// TIA Portal V20 export
ORGANIZATION_BLOCK "Main"   // OB1, LAD, ProgramCycle
TITLE = "Main Program Sweep (Cycle)"
{ S7_Optimized_Access := 'TRUE' }
// stored: SetENOAutomatically false
   VAR_INPUT
      Initial_Call : Bool;   // Initial call of this OB
      Remanence : Bool;   // =True, if remanent data are available
   END_VAR
BEGIN

REGION Network 1
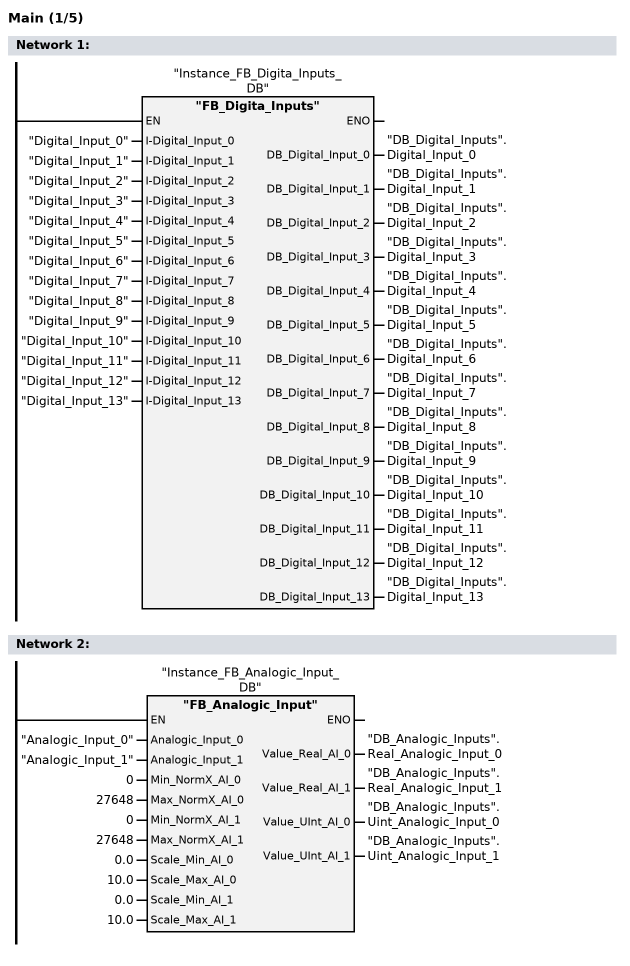
   RUNG wire#powerrail
      "Instance_FB_Digita_Inputs_DB"("I-Digital_Input_0" := "Digital_Input_0", "I-Digital_Input_1" := "Digital_Input_1", "I-Digital_Input_2" := "Digital_Input_2", "I-Digital_Input_3" := "Digital_Input_3", "I-Digital_Input_4" := "Digital_Input_4", "I-Digital_Input_5" := "Digital_Input_5", "I-Digital_Input_6" := "Digital_Input_6", "I-Digital_Input_7" := "Digital_Input_7", "I-Digital_Input_8" := "Digital_Input_8", "I-Digital_Input_9" := "Digital_Input_9", "I-Digital_Input_10" := "Digital_Input_10", "I-Digital_Input_11" := "Digital_Input_11", "I-Digital_Input_12" := "Digital_Input_12", "I-Digital_Input_13" := "Digital_Input_13", DB_Digital_Input_0 => "DB_Digital_Inputs".Digital_Input_0, DB_Digital_Input_1 => "DB_Digital_Inputs".Digital_Input_1, DB_Digital_Input_2 => "DB_Digital_Inputs".Digital_Input_2, DB_Digital_Input_3 => "DB_Digital_Inputs".Digital_Input_3, DB_Digital_Input_4 => "DB_Digital_Inputs".Digital_Input_4, DB_Digital_Input_5 => "DB_Digital_Inputs".Digital_Input_5, DB_Digital_Input_6 => "DB_Digital_Inputs".Digital_Input_6, DB_Digital_Input_7 => "DB_Digital_Inputs".Digital_Input_7, DB_Digital_Input_8 => "DB_Digital_Inputs".Digital_Input_8, DB_Digital_Input_9 => "DB_Digital_Inputs".Digital_Input_9, DB_Digital_Input_10 => "DB_Digital_Inputs".Digital_Input_10, DB_Digital_Input_11 => "DB_Digital_Inputs".Digital_Input_11, DB_Digital_Input_12 => "DB_Digital_Inputs".Digital_Input_12, DB_Digital_Input_13 => "DB_Digital_Inputs".Digital_Input_13)
   END_RUNG
   // the same network as SCL:
   "Instance_FB_Digita_Inputs_DB"("I-Digital_Input_0" := "Digital_Input_0",   // "FB_Digita_Inputs"
                           "I-Digital_Input_1" := "Digital_Input_1",
                           "I-Digital_Input_2" := "Digital_Input_2",
                           "I-Digital_Input_3" := "Digital_Input_3",
                           "I-Digital_Input_4" := "Digital_Input_4",
                           "I-Digital_Input_5" := "Digital_Input_5",
                           "I-Digital_Input_6" := "Digital_Input_6",
                           "I-Digital_Input_7" := "Digital_Input_7",
                           "I-Digital_Input_8" := "Digital_Input_8",
                           "I-Digital_Input_9" := "Digital_Input_9",
                           "I-Digital_Input_10" := "Digital_Input_10",
                           "I-Digital_Input_11" := "Digital_Input_11",
                           "I-Digital_Input_12" := "Digital_Input_12",
                           "I-Digital_Input_13" := "Digital_Input_13",
                           DB_Digital_Input_0 => "DB_Digital_Inputs".Digital_Input_0,
                           DB_Digital_Input_1 => "DB_Digital_Inputs".Digital_Input_1,
                           DB_Digital_Input_2 => "DB_Digital_Inputs".Digital_Input_2,
                           DB_Digital_Input_3 => "DB_Digital_Inputs".Digital_Input_3,
                           DB_Digital_Input_4 => "DB_Digital_Inputs".Digital_Input_4,
                           DB_Digital_Input_5 => "DB_Digital_Inputs".Digital_Input_5,
                           DB_Digital_Input_6 => "DB_Digital_Inputs".Digital_Input_6,
                           DB_Digital_Input_7 => "DB_Digital_Inputs".Digital_Input_7,
                           DB_Digital_Input_8 => "DB_Digital_Inputs".Digital_Input_8,
                           DB_Digital_Input_9 => "DB_Digital_Inputs".Digital_Input_9,
                           DB_Digital_Input_10 => "DB_Digital_Inputs".Digital_Input_10,
                           DB_Digital_Input_11 => "DB_Digital_Inputs".Digital_Input_11,
                           DB_Digital_Input_12 => "DB_Digital_Inputs".Digital_Input_12,
                           DB_Digital_Input_13 => "DB_Digital_Inputs".Digital_Input_13);
END_REGION

REGION Network 2
   RUNG wire#powerrail
      "Instance_FB_Analogic_Input_DB"(Analogic_Input_0 := "Analogic_Input_0", Analogic_Input_1 := "Analogic_Input_1", Min_NormX_AI_0 := 0, Max_NormX_AI_0 := 27648, Min_NormX_AI_1 := 0, Max_NormX_AI_1 := 27648, Scale_Min_AI_0 := 0.0, Scale_Max_AI_0 := 10.0, Scale_Min_AI_1 := 0.0, Scale_Max_AI_1 := 10.0, Value_Real_AI_0 => "DB_Analogic_Inputs".Real_Analogic_Input_0, Value_Real_AI_1 => "DB_Analogic_Inputs".Real_Analogic_Input_1, Value_UInt_AI_0 => "DB_Analogic_Inputs".Uint_Analogic_Input_0, Value_UInt_AI_1 => "DB_Analogic_Inputs".Uint_Analogic_Input_1)
   END_RUNG
   // the same network as SCL:
   "Instance_FB_Analogic_Input_DB"(Analogic_Input_0 := "Analogic_Input_0",   // "FB_Analogic_Input"
                           Analogic_Input_1 := "Analogic_Input_1",
                           Min_NormX_AI_0 := 0,
                           Max_NormX_AI_0 := 27648,
                           Min_NormX_AI_1 := 0,
                           Max_NormX_AI_1 := 27648,
                           Scale_Min_AI_0 := 0.0,
                           Scale_Max_AI_0 := 10.0,
                           Scale_Min_AI_1 := 0.0,
                           Scale_Max_AI_1 := 10.0,
                           Value_Real_AI_0 => "DB_Analogic_Inputs".Real_Analogic_Input_0,
                           Value_Real_AI_1 => "DB_Analogic_Inputs".Real_Analogic_Input_1,
                           Value_UInt_AI_0 => "DB_Analogic_Inputs".Uint_Analogic_Input_0,
                           Value_UInt_AI_1 => "DB_Analogic_Inputs".Uint_Analogic_Input_1);
END_REGION

REGION Network 3
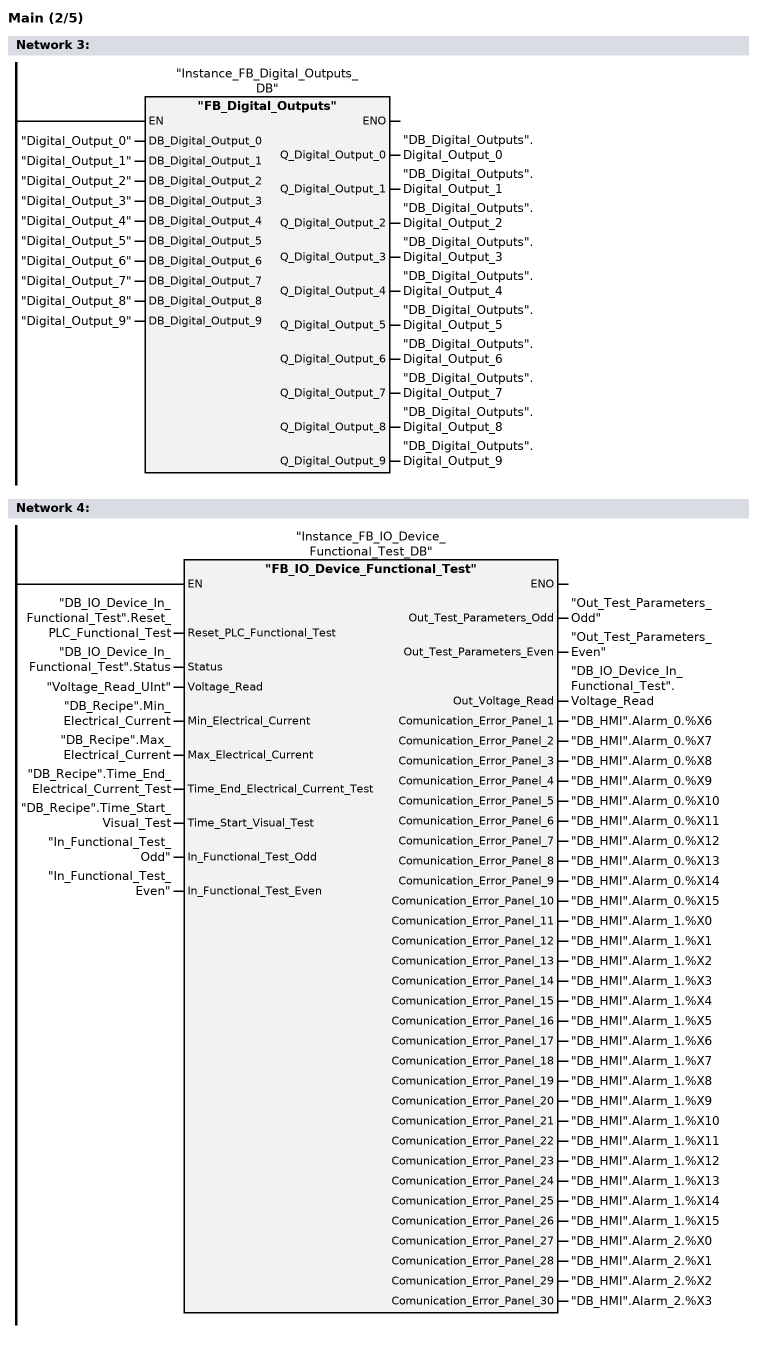
   RUNG wire#powerrail
      "Instance_FB_Digital_Outputs_DB"(DB_Digital_Output_0 := "Digital_Output_0", DB_Digital_Output_1 := "Digital_Output_1", DB_Digital_Output_2 := "Digital_Output_2", DB_Digital_Output_3 := "Digital_Output_3", DB_Digital_Output_4 := "Digital_Output_4", DB_Digital_Output_5 := "Digital_Output_5", DB_Digital_Output_6 := "Digital_Output_6", DB_Digital_Output_7 := "Digital_Output_7", DB_Digital_Output_8 := "Digital_Output_8", DB_Digital_Output_9 := "Digital_Output_9", Q_Digital_Output_0 => "DB_Digital_Outputs".Digital_Output_0, Q_Digital_Output_1 => "DB_Digital_Outputs".Digital_Output_1, Q_Digital_Output_2 => "DB_Digital_Outputs".Digital_Output_2, Q_Digital_Output_3 => "DB_Digital_Outputs".Digital_Output_3, Q_Digital_Output_4 => "DB_Digital_Outputs".Digital_Output_4, Q_Digital_Output_5 => "DB_Digital_Outputs".Digital_Output_5, Q_Digital_Output_6 => "DB_Digital_Outputs".Digital_Output_6, Q_Digital_Output_7 => "DB_Digital_Outputs".Digital_Output_7, Q_Digital_Output_8 => "DB_Digital_Outputs".Digital_Output_8, Q_Digital_Output_9 => "DB_Digital_Outputs".Digital_Output_9)
   END_RUNG
   // the same network as SCL:
   "Instance_FB_Digital_Outputs_DB"(DB_Digital_Output_0 := "Digital_Output_0",   // "FB_Digital_Outputs"
                           DB_Digital_Output_1 := "Digital_Output_1",
                           DB_Digital_Output_2 := "Digital_Output_2",
                           DB_Digital_Output_3 := "Digital_Output_3",
                           DB_Digital_Output_4 := "Digital_Output_4",
                           DB_Digital_Output_5 := "Digital_Output_5",
                           DB_Digital_Output_6 := "Digital_Output_6",
                           DB_Digital_Output_7 := "Digital_Output_7",
                           DB_Digital_Output_8 := "Digital_Output_8",
                           DB_Digital_Output_9 := "Digital_Output_9",
                           Q_Digital_Output_0 => "DB_Digital_Outputs".Digital_Output_0,
                           Q_Digital_Output_1 => "DB_Digital_Outputs".Digital_Output_1,
                           Q_Digital_Output_2 => "DB_Digital_Outputs".Digital_Output_2,
                           Q_Digital_Output_3 => "DB_Digital_Outputs".Digital_Output_3,
                           Q_Digital_Output_4 => "DB_Digital_Outputs".Digital_Output_4,
                           Q_Digital_Output_5 => "DB_Digital_Outputs".Digital_Output_5,
                           Q_Digital_Output_6 => "DB_Digital_Outputs".Digital_Output_6,
                           Q_Digital_Output_7 => "DB_Digital_Outputs".Digital_Output_7,
                           Q_Digital_Output_8 => "DB_Digital_Outputs".Digital_Output_8,
                           Q_Digital_Output_9 => "DB_Digital_Outputs".Digital_Output_9);
END_REGION

REGION Network 4
   RUNG wire#powerrail
      "Instance_FB_IO_Device_Functional_Test_DB"(Reset_PLC_Functional_Test := "DB_IO_Device_In_Functional_Test".Reset_PLC_Functional_Test, Status := "DB_IO_Device_In_Functional_Test".Status, Voltage_Read := "Voltage_Read_UInt", Min_Electrical_Current := "DB_Recipe".Min_Electrical_Current, Max_Electrical_Current := "DB_Recipe".Max_Electrical_Current, Time_End_Electrical_Current_Test := "DB_Recipe".Time_End_Electrical_Current_Test, Time_Start_Visual_Test := "DB_Recipe".Time_Start_Visual_Test, In_Functional_Test_Odd := "In_Functional_Test_Odd", In_Functional_Test_Even := "In_Functional_Test_Even", Out_Test_Parameters_Odd => "Out_Test_Parameters_Odd", Out_Test_Parameters_Even => "Out_Test_Parameters_Even", Out_Voltage_Read => "DB_IO_Device_In_Functional_Test".Voltage_Read, Comunication_Error_Panel_1 => "DB_HMI".Alarm_0.%X6, Comunication_Error_Panel_2 => "DB_HMI".Alarm_0.%X7, Comunication_Error_Panel_3 => "DB_HMI".Alarm_0.%X8, Comunication_Error_Panel_4 => "DB_HMI".Alarm_0.%X9, Comunication_Error_Panel_5 => "DB_HMI".Alarm_0.%X10, Comunication_Error_Panel_6 => "DB_HMI".Alarm_0.%X11, Comunication_Error_Panel_7 => "DB_HMI".Alarm_0.%X12, Comunication_Error_Panel_8 => "DB_HMI".Alarm_0.%X13, Comunication_Error_Panel_9 => "DB_HMI".Alarm_0.%X14, Comunication_Error_Panel_10 => "DB_HMI".Alarm_0.%X15, Comunication_Error_Panel_11 => "DB_HMI".Alarm_1.%X0, Comunication_Error_Panel_12 => "DB_HMI".Alarm_1.%X1, Comunication_Error_Panel_13 => "DB_HMI".Alarm_1.%X2, Comunication_Error_Panel_14 => "DB_HMI".Alarm_1.%X3, Comunication_Error_Panel_15 => "DB_HMI".Alarm_1.%X4, Comunication_Error_Panel_16 => "DB_HMI".Alarm_1.%X5, Comunication_Error_Panel_17 => "DB_HMI".Alarm_1.%X6, Comunication_Error_Panel_18 => "DB_HMI".Alarm_1.%X7, Comunication_Error_Panel_19 => "DB_HMI".Alarm_1.%X8, Comunication_Error_Panel_20 => "DB_HMI".Alarm_1.%X9, Comunication_Error_Panel_21 => "DB_HMI".Alarm_1.%X10, Comunication_Error_Panel_22 => "DB_HMI".Alarm_1.%X11, Comunication_Error_Panel_23 => "DB_HMI".Alarm_1.%X12, Comunication_Error_Panel_24 => "DB_HMI".Alarm_1.%X13, Comunication_Error_Panel_25 => "DB_HMI".Alarm_1.%X14, Comunication_Error_Panel_26 => "DB_HMI".Alarm_1.%X15, Comunication_Error_Panel_27 => "DB_HMI".Alarm_2.%X0, Comunication_Error_Panel_28 => "DB_HMI".Alarm_2.%X1, Comunication_Error_Panel_29 => "DB_HMI".Alarm_2.%X2, Comunication_Error_Panel_30 => "DB_HMI".Alarm_2.%X3)
   END_RUNG
   // the same network as SCL:
   "Instance_FB_IO_Device_Functional_Test_DB"(Reset_PLC_Functional_Test := "DB_IO_Device_In_Functional_Test".Reset_PLC_Functional_Test,   // "FB_IO_Device_Functional_Test"
                           Status := "DB_IO_Device_In_Functional_Test".Status,
                           Voltage_Read := "Voltage_Read_UInt",
                           Min_Electrical_Current := "DB_Recipe".Min_Electrical_Current,
                           Max_Electrical_Current := "DB_Recipe".Max_Electrical_Current,
                           Time_End_Electrical_Current_Test := "DB_Recipe".Time_End_Electrical_Current_Test,
                           Time_Start_Visual_Test := "DB_Recipe".Time_Start_Visual_Test,
                           In_Functional_Test_Odd := "In_Functional_Test_Odd",
                           In_Functional_Test_Even := "In_Functional_Test_Even",
                           Out_Test_Parameters_Odd => "Out_Test_Parameters_Odd",
                           Out_Test_Parameters_Even => "Out_Test_Parameters_Even",
                           Out_Voltage_Read => "DB_IO_Device_In_Functional_Test".Voltage_Read,
                           Comunication_Error_Panel_1 => "DB_HMI".Alarm_0.%X6,
                           Comunication_Error_Panel_2 => "DB_HMI".Alarm_0.%X7,
                           Comunication_Error_Panel_3 => "DB_HMI".Alarm_0.%X8,
                           Comunication_Error_Panel_4 => "DB_HMI".Alarm_0.%X9,
                           Comunication_Error_Panel_5 => "DB_HMI".Alarm_0.%X10,
                           Comunication_Error_Panel_6 => "DB_HMI".Alarm_0.%X11,
                           Comunication_Error_Panel_7 => "DB_HMI".Alarm_0.%X12,
                           Comunication_Error_Panel_8 => "DB_HMI".Alarm_0.%X13,
                           Comunication_Error_Panel_9 => "DB_HMI".Alarm_0.%X14,
                           Comunication_Error_Panel_10 => "DB_HMI".Alarm_0.%X15,
                           Comunication_Error_Panel_11 => "DB_HMI".Alarm_1.%X0,
                           Comunication_Error_Panel_12 => "DB_HMI".Alarm_1.%X1,
                           Comunication_Error_Panel_13 => "DB_HMI".Alarm_1.%X2,
                           Comunication_Error_Panel_14 => "DB_HMI".Alarm_1.%X3,
                           Comunication_Error_Panel_15 => "DB_HMI".Alarm_1.%X4,
                           Comunication_Error_Panel_16 => "DB_HMI".Alarm_1.%X5,
                           Comunication_Error_Panel_17 => "DB_HMI".Alarm_1.%X6,
                           Comunication_Error_Panel_18 => "DB_HMI".Alarm_1.%X7,
                           Comunication_Error_Panel_19 => "DB_HMI".Alarm_1.%X8,
                           Comunication_Error_Panel_20 => "DB_HMI".Alarm_1.%X9,
                           Comunication_Error_Panel_21 => "DB_HMI".Alarm_1.%X10,
                           Comunication_Error_Panel_22 => "DB_HMI".Alarm_1.%X11,
                           Comunication_Error_Panel_23 => "DB_HMI".Alarm_1.%X12,
                           Comunication_Error_Panel_24 => "DB_HMI".Alarm_1.%X13,
                           Comunication_Error_Panel_25 => "DB_HMI".Alarm_1.%X14,
                           Comunication_Error_Panel_26 => "DB_HMI".Alarm_1.%X15,
                           Comunication_Error_Panel_27 => "DB_HMI".Alarm_2.%X0,
                           Comunication_Error_Panel_28 => "DB_HMI".Alarm_2.%X1,
                           Comunication_Error_Panel_29 => "DB_HMI".Alarm_2.%X2,
                           Comunication_Error_Panel_30 => "DB_HMI".Alarm_2.%X3);
END_REGION

REGION Network 5
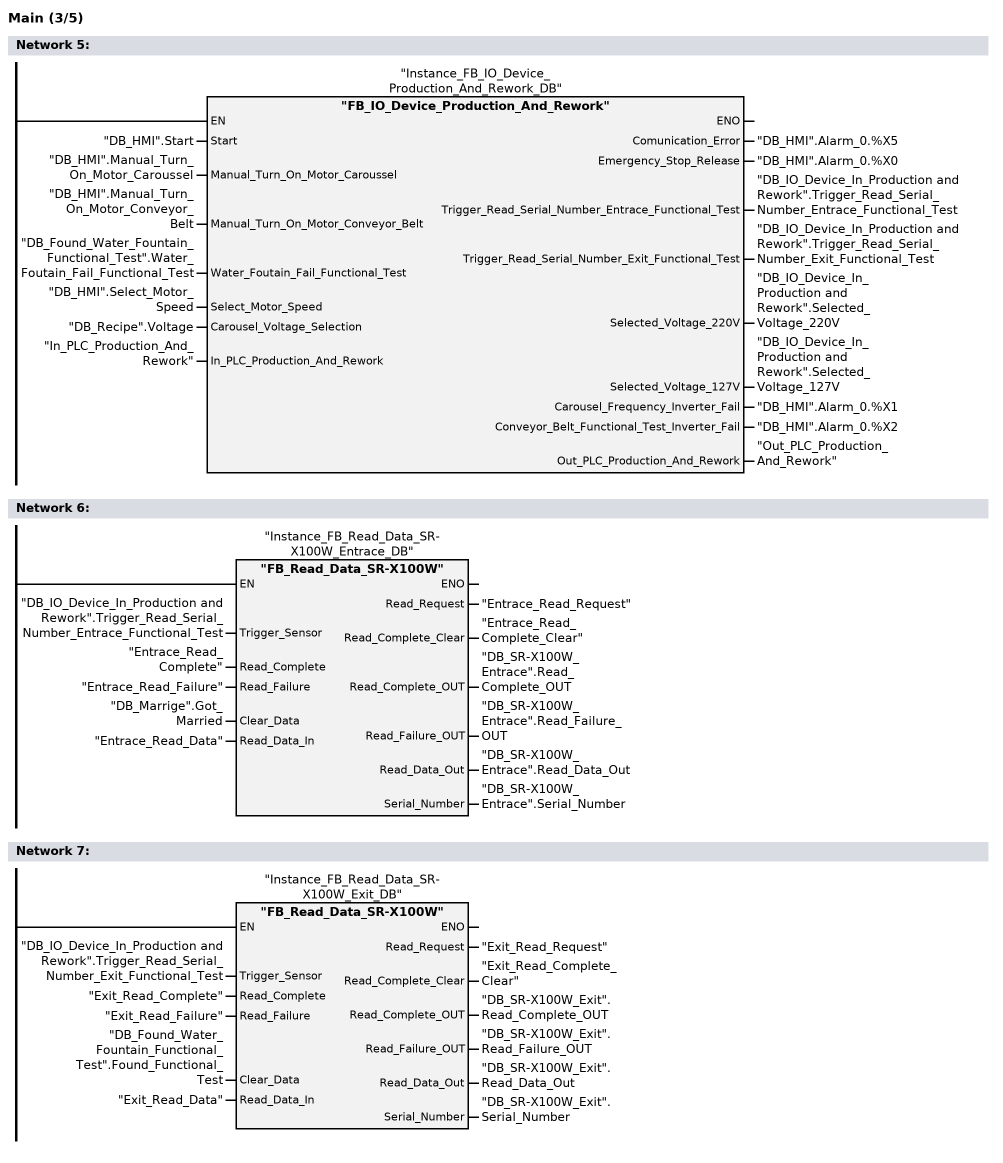
   RUNG wire#powerrail
      "Instance_FB_IO_Device_Production_And_Rework_DB"(Start := "DB_HMI".Start, Manual_Turn_On_Motor_Caroussel := "DB_HMI".Manual_Turn_On_Motor_Caroussel, Manual_Turn_On_Motor_Conveyor_Belt := "DB_HMI".Manual_Turn_On_Motor_Conveyor_Belt, Water_Foutain_Fail_Functional_Test := "DB_Found_Water_Fountain_Functional_Test".Water_Foutain_Fail_Functional_Test, Select_Motor_Speed := "DB_HMI".Select_Motor_Speed, Carousel_Voltage_Selection := "DB_Recipe".Voltage, In_PLC_Production_And_Rework := "In_PLC_Production_And_Rework", Comunication_Error => "DB_HMI".Alarm_0.%X5, Emergency_Stop_Release => "DB_HMI".Alarm_0.%X0, Trigger_Read_Serial_Number_Entrace_Functional_Test => "DB_IO_Device_In_Production and Rework".Trigger_Read_Serial_Number_Entrace_Functional_Test, Trigger_Read_Serial_Number_Exit_Functional_Test => "DB_IO_Device_In_Production and Rework".Trigger_Read_Serial_Number_Exit_Functional_Test, Selected_Voltage_220V => "DB_IO_Device_In_Production and Rework".Selected_Voltage_220V, Selected_Voltage_127V => "DB_IO_Device_In_Production and Rework".Selected_Voltage_127V, Carousel_Frequency_Inverter_Fail => "DB_HMI".Alarm_0.%X1, Conveyor_Belt_Functional_Test_Inverter_Fail => "DB_HMI".Alarm_0.%X2, Out_PLC_Production_And_Rework => "Out_PLC_Production_And_Rework")
   END_RUNG
   // the same network as SCL:
   "Instance_FB_IO_Device_Production_And_Rework_DB"(Start := "DB_HMI".Start,   // "FB_IO_Device_Production_And_Rework"
                           Manual_Turn_On_Motor_Caroussel := "DB_HMI".Manual_Turn_On_Motor_Caroussel,
                           Manual_Turn_On_Motor_Conveyor_Belt := "DB_HMI".Manual_Turn_On_Motor_Conveyor_Belt,
                           Water_Foutain_Fail_Functional_Test := "DB_Found_Water_Fountain_Functional_Test".Water_Foutain_Fail_Functional_Test,
                           Select_Motor_Speed := "DB_HMI".Select_Motor_Speed,
                           Carousel_Voltage_Selection := "DB_Recipe".Voltage,
                           In_PLC_Production_And_Rework := "In_PLC_Production_And_Rework",
                           Comunication_Error => "DB_HMI".Alarm_0.%X5,
                           Emergency_Stop_Release => "DB_HMI".Alarm_0.%X0,
                           Trigger_Read_Serial_Number_Entrace_Functional_Test => "DB_IO_Device_In_Production and Rework".Trigger_Read_Serial_Number_Entrace_Functional_Test,
                           Trigger_Read_Serial_Number_Exit_Functional_Test => "DB_IO_Device_In_Production and Rework".Trigger_Read_Serial_Number_Exit_Functional_Test,
                           Selected_Voltage_220V => "DB_IO_Device_In_Production and Rework".Selected_Voltage_220V,
                           Selected_Voltage_127V => "DB_IO_Device_In_Production and Rework".Selected_Voltage_127V,
                           Carousel_Frequency_Inverter_Fail => "DB_HMI".Alarm_0.%X1,
                           Conveyor_Belt_Functional_Test_Inverter_Fail => "DB_HMI".Alarm_0.%X2,
                           Out_PLC_Production_And_Rework => "Out_PLC_Production_And_Rework");
END_REGION

REGION Network 6
   RUNG wire#powerrail
      "Instance_FB_Read_Data_SR-X100W_Entrace_DB"(Trigger_Sensor := "DB_IO_Device_In_Production and Rework".Trigger_Read_Serial_Number_Entrace_Functional_Test, Read_Complete := "Entrace_Read_Complete", Read_Failure := "Entrace_Read_Failure", Clear_Data := "DB_Marrige".Got_Married, Read_Data_In := "Entrace_Read_Data", Read_Request => "Entrace_Read_Request", Read_Complete_Clear => "Entrace_Read_Complete_Clear", Read_Complete_OUT => "DB_SR-X100W_Entrace".Read_Complete_OUT, Read_Failure_OUT => "DB_SR-X100W_Entrace".Read_Failure_OUT, Read_Data_Out => "DB_SR-X100W_Entrace".Read_Data_Out, Serial_Number => "DB_SR-X100W_Entrace".Serial_Number)
   END_RUNG
   // the same network as SCL:
   "Instance_FB_Read_Data_SR-X100W_Entrace_DB"(Trigger_Sensor := "DB_IO_Device_In_Production and Rework".Trigger_Read_Serial_Number_Entrace_Functional_Test,   // "FB_Read_Data_SR-X100W"
                           Read_Complete := "Entrace_Read_Complete",
                           Read_Failure := "Entrace_Read_Failure",
                           Clear_Data := "DB_Marrige".Got_Married,
                           Read_Data_In := "Entrace_Read_Data",
                           Read_Request => "Entrace_Read_Request",
                           Read_Complete_Clear => "Entrace_Read_Complete_Clear",
                           Read_Complete_OUT => "DB_SR-X100W_Entrace".Read_Complete_OUT,
                           Read_Failure_OUT => "DB_SR-X100W_Entrace".Read_Failure_OUT,
                           Read_Data_Out => "DB_SR-X100W_Entrace".Read_Data_Out,
                           Serial_Number => "DB_SR-X100W_Entrace".Serial_Number);
END_REGION

REGION Network 7
   RUNG wire#powerrail
      "Instance_FB_Read_Data_SR-X100W_Exit_DB"(Trigger_Sensor := "DB_IO_Device_In_Production and Rework".Trigger_Read_Serial_Number_Exit_Functional_Test, Read_Complete := "Exit_Read_Complete", Read_Failure := "Exit_Read_Failure", Clear_Data := "DB_Found_Water_Fountain_Functional_Test".Found_Functional_Test, Read_Data_In := "Exit_Read_Data", Read_Request => "Exit_Read_Request", Read_Complete_Clear => "Exit_Read_Complete_Clear", Read_Complete_OUT => "DB_SR-X100W_Exit".Read_Complete_OUT, Read_Failure_OUT => "DB_SR-X100W_Exit".Read_Failure_OUT, Read_Data_Out => "DB_SR-X100W_Exit".Read_Data_Out, Serial_Number => "DB_SR-X100W_Exit".Serial_Number)
   END_RUNG
   // the same network as SCL:
   "Instance_FB_Read_Data_SR-X100W_Exit_DB"(Trigger_Sensor := "DB_IO_Device_In_Production and Rework".Trigger_Read_Serial_Number_Exit_Functional_Test,   // "FB_Read_Data_SR-X100W"
                           Read_Complete := "Exit_Read_Complete",
                           Read_Failure := "Exit_Read_Failure",
                           Clear_Data := "DB_Found_Water_Fountain_Functional_Test".Found_Functional_Test,
                           Read_Data_In := "Exit_Read_Data",
                           Read_Request => "Exit_Read_Request",
                           Read_Complete_Clear => "Exit_Read_Complete_Clear",
                           Read_Complete_OUT => "DB_SR-X100W_Exit".Read_Complete_OUT,
                           Read_Failure_OUT => "DB_SR-X100W_Exit".Read_Failure_OUT,
                           Read_Data_Out => "DB_SR-X100W_Exit".Read_Data_Out,
                           Serial_Number => "DB_SR-X100W_Exit".Serial_Number);
END_REGION

REGION Network 8
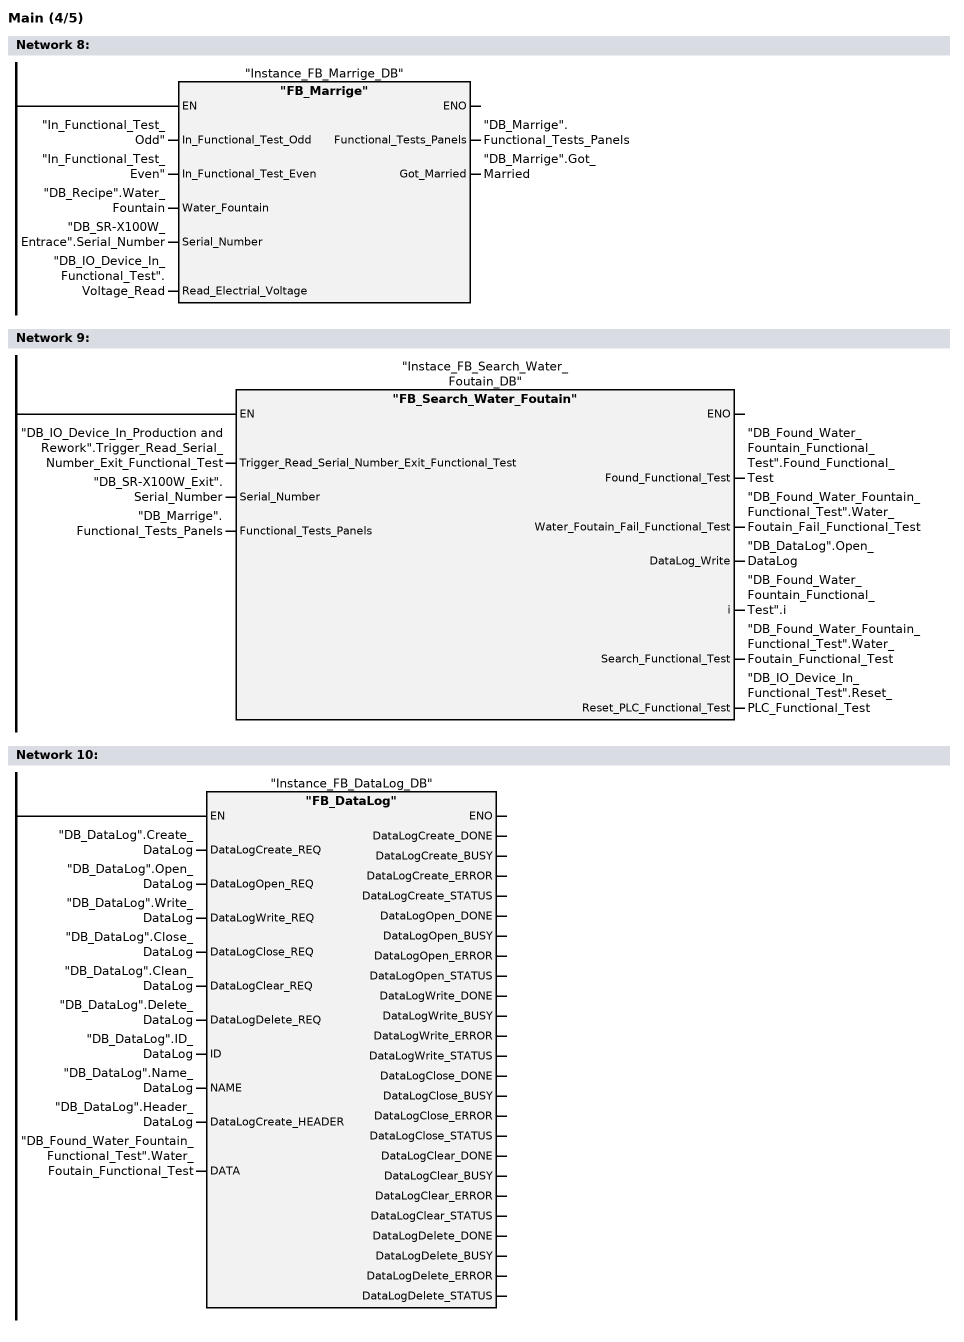
   RUNG wire#powerrail
      "Instance_FB_Marrige_DB"(In_Functional_Test_Odd := "In_Functional_Test_Odd", In_Functional_Test_Even := "In_Functional_Test_Even", Water_Fountain := "DB_Recipe".Water_Fountain, Serial_Number := "DB_SR-X100W_Entrace".Serial_Number, Read_Electrial_Voltage := "DB_IO_Device_In_Functional_Test".Voltage_Read, Functional_Tests_Panels => "DB_Marrige".Functional_Tests_Panels, Got_Married => "DB_Marrige".Got_Married)
   END_RUNG
   // the same network as SCL:
   "Instance_FB_Marrige_DB"(In_Functional_Test_Odd := "In_Functional_Test_Odd",   // "FB_Marrige"
                           In_Functional_Test_Even := "In_Functional_Test_Even",
                           Water_Fountain := "DB_Recipe".Water_Fountain,
                           Serial_Number := "DB_SR-X100W_Entrace".Serial_Number,
                           Read_Electrial_Voltage := "DB_IO_Device_In_Functional_Test".Voltage_Read,
                           Functional_Tests_Panels => "DB_Marrige".Functional_Tests_Panels,
                           Got_Married => "DB_Marrige".Got_Married);
END_REGION

REGION Network 9
   RUNG wire#powerrail
      "Instace_FB_Search_Water_Foutain_DB"(Trigger_Read_Serial_Number_Exit_Functional_Test := "DB_IO_Device_In_Production and Rework".Trigger_Read_Serial_Number_Exit_Functional_Test, Serial_Number := "DB_SR-X100W_Exit".Serial_Number, Functional_Tests_Panels := "DB_Marrige".Functional_Tests_Panels, Found_Functional_Test => "DB_Found_Water_Fountain_Functional_Test".Found_Functional_Test, Water_Foutain_Fail_Functional_Test => "DB_Found_Water_Fountain_Functional_Test".Water_Foutain_Fail_Functional_Test, DataLog_Write => "DB_DataLog".Open_DataLog, i => "DB_Found_Water_Fountain_Functional_Test".i, Search_Functional_Test => "DB_Found_Water_Fountain_Functional_Test".Water_Foutain_Functional_Test, Reset_PLC_Functional_Test => "DB_IO_Device_In_Functional_Test".Reset_PLC_Functional_Test)
   END_RUNG
   // the same network as SCL:
   "Instace_FB_Search_Water_Foutain_DB"(Trigger_Read_Serial_Number_Exit_Functional_Test := "DB_IO_Device_In_Production and Rework".Trigger_Read_Serial_Number_Exit_Functional_Test,   // "FB_Search_Water_Foutain"
                           Serial_Number := "DB_SR-X100W_Exit".Serial_Number,
                           Functional_Tests_Panels := "DB_Marrige".Functional_Tests_Panels,
                           Found_Functional_Test => "DB_Found_Water_Fountain_Functional_Test".Found_Functional_Test,
                           Water_Foutain_Fail_Functional_Test => "DB_Found_Water_Fountain_Functional_Test".Water_Foutain_Fail_Functional_Test,
                           DataLog_Write => "DB_DataLog".Open_DataLog,
                           i => "DB_Found_Water_Fountain_Functional_Test".i,
                           Search_Functional_Test => "DB_Found_Water_Fountain_Functional_Test".Water_Foutain_Functional_Test,
                           Reset_PLC_Functional_Test => "DB_IO_Device_In_Functional_Test".Reset_PLC_Functional_Test);
END_REGION

REGION Network 10
   RUNG wire#powerrail
      "Instance_FB_DataLog_DB"(DataLogCreate_REQ := "DB_DataLog".Create_DataLog, DataLogOpen_REQ := "DB_DataLog".Open_DataLog, DataLogWrite_REQ := "DB_DataLog".Write_DataLog, DataLogClose_REQ := "DB_DataLog".Close_DataLog, DataLogClear_REQ := "DB_DataLog".Clean_DataLog, DataLogDelete_REQ := "DB_DataLog".Delete_DataLog, ID := "DB_DataLog".ID_DataLog, "NAME" := "DB_DataLog".Name_DataLog, DataLogCreate_HEADER := "DB_DataLog".Header_DataLog, DATA := "DB_Found_Water_Fountain_Functional_Test".Water_Foutain_Functional_Test, DataLogCreate_DONE =>, DataLogCreate_BUSY =>, DataLogCreate_ERROR =>, DataLogCreate_STATUS =>, DataLogOpen_DONE =>, DataLogOpen_BUSY =>, DataLogOpen_ERROR =>, DataLogOpen_STATUS =>, DataLogWrite_DONE =>, DataLogWrite_BUSY =>, DataLogWrite_ERROR =>, DataLogWrite_STATUS =>, DataLogClose_DONE =>, DataLogClose_BUSY =>, DataLogClose_ERROR =>, DataLogClose_STATUS =>, DataLogClear_DONE =>, DataLogClear_BUSY =>, DataLogClear_ERROR =>, DataLogClear_STATUS =>, DataLogDelete_DONE =>, DataLogDelete_BUSY =>, DataLogDelete_ERROR =>, DataLogDelete_STATUS =>)
   END_RUNG
   // the same network as SCL:
   "Instance_FB_DataLog_DB"(DataLogCreate_REQ := "DB_DataLog".Create_DataLog,   // "FB_DataLog"
                           DataLogOpen_REQ := "DB_DataLog".Open_DataLog,
                           DataLogWrite_REQ := "DB_DataLog".Write_DataLog,
                           DataLogClose_REQ := "DB_DataLog".Close_DataLog,
                           DataLogClear_REQ := "DB_DataLog".Clean_DataLog,
                           DataLogDelete_REQ := "DB_DataLog".Delete_DataLog,
                           ID := "DB_DataLog".ID_DataLog,
                           "NAME" := "DB_DataLog".Name_DataLog,
                           DataLogCreate_HEADER := "DB_DataLog".Header_DataLog,
                           DATA := "DB_Found_Water_Fountain_Functional_Test".Water_Foutain_Functional_Test);
END_REGION

REGION Network 11
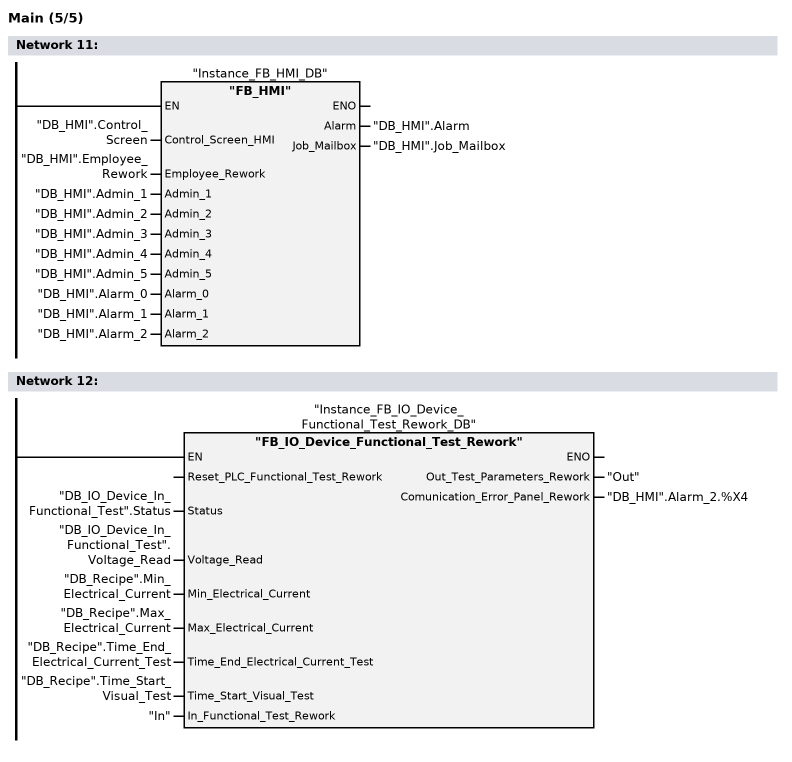
   RUNG wire#powerrail
      "Instance_FB_HMI_DB"(Control_Screen_HMI := "DB_HMI".Control_Screen, Employee_Rework := "DB_HMI".Employee_Rework, Admin_1 := "DB_HMI".Admin_1, Admin_2 := "DB_HMI".Admin_2, Admin_3 := "DB_HMI".Admin_3, Admin_4 := "DB_HMI".Admin_4, Admin_5 := "DB_HMI".Admin_5, Alarm_0 := "DB_HMI".Alarm_0, Alarm_1 := "DB_HMI".Alarm_1, Alarm_2 := "DB_HMI".Alarm_2, Alarm => "DB_HMI".Alarm, Job_Mailbox => "DB_HMI".Job_Mailbox)
   END_RUNG
   // the same network as SCL:
   "Instance_FB_HMI_DB"(Control_Screen_HMI := "DB_HMI".Control_Screen,   // "FB_HMI"
                        Employee_Rework := "DB_HMI".Employee_Rework,
                        Admin_1 := "DB_HMI".Admin_1,
                        Admin_2 := "DB_HMI".Admin_2,
                        Admin_3 := "DB_HMI".Admin_3,
                        Admin_4 := "DB_HMI".Admin_4,
                        Admin_5 := "DB_HMI".Admin_5,
                        Alarm_0 := "DB_HMI".Alarm_0,
                        Alarm_1 := "DB_HMI".Alarm_1,
                        Alarm_2 := "DB_HMI".Alarm_2,
                        Alarm => "DB_HMI".Alarm,
                        Job_Mailbox => "DB_HMI".Job_Mailbox);
END_REGION

REGION Network 12
   RUNG wire#powerrail
      "Instance_FB_IO_Device_Functional_Test_Rework_DB"(Reset_PLC_Functional_Test_Rework :=, Status := "DB_IO_Device_In_Functional_Test".Status, Voltage_Read := "DB_IO_Device_In_Functional_Test".Voltage_Read, Min_Electrical_Current := "DB_Recipe".Min_Electrical_Current, Max_Electrical_Current := "DB_Recipe".Max_Electrical_Current, Time_End_Electrical_Current_Test := "DB_Recipe".Time_End_Electrical_Current_Test, Time_Start_Visual_Test := "DB_Recipe".Time_Start_Visual_Test, In_Functional_Test_Rework := "In", Out_Test_Parameters_Rework => "Out", Comunication_Error_Panel_Rework => "DB_HMI".Alarm_2.%X4)
   END_RUNG
   // the same network as SCL:
   "Instance_FB_IO_Device_Functional_Test_Rework_DB"(Status := "DB_IO_Device_In_Functional_Test".Status,   // "FB_IO_Device_Functional_Test_Rework"
                           Voltage_Read := "DB_IO_Device_In_Functional_Test".Voltage_Read,
                           Min_Electrical_Current := "DB_Recipe".Min_Electrical_Current,
                           Max_Electrical_Current := "DB_Recipe".Max_Electrical_Current,
                           Time_End_Electrical_Current_Test := "DB_Recipe".Time_End_Electrical_Current_Test,
                           Time_Start_Visual_Test := "DB_Recipe".Time_Start_Visual_Test,
                           In_Functional_Test_Rework := "In",
                           Out_Test_Parameters_Rework => "Out",
                           Comunication_Error_Panel_Rework => "DB_HMI".Alarm_2.%X4);
END_REGION
END_ORGANIZATION_BLOCK
